// SIMATIC S7-200 project (STEP 7-Micro/WIN), CPU 221 REL 01.10

SYMBOL_TABLE USER1
BT               I0.0     // dieu khien bang tay
TD               I0.1     // dieu khien tu dong
s1               I0.2     // nut giu mo cong
s3               I0.3     // cong tac hanh trinh mo cong
s2               I0.4     // nut giu dong cong
s4               I0.5     // cong tac hanh trinh dong cong
open             I0.6     // mo cua o che do tu dong
close            I0.7     // dong cua o che do tu dong
s5               I1.0     // dung he thong
CDBT             Q0.0     // che do bang tay
CDTD             Q0.1     // che do tu dong
MT               Q0.2     // mo cong
MN               Q0.3     // dong cong
H1               Q0.4     // den bao
s6               I1.1     // dole nhiet dung he thong
END_SYMBOL_TABLE

ORGANIZATION_BLOCK MAIN:OB1
TITLE=PROGRAM COMMENTS
BEGIN
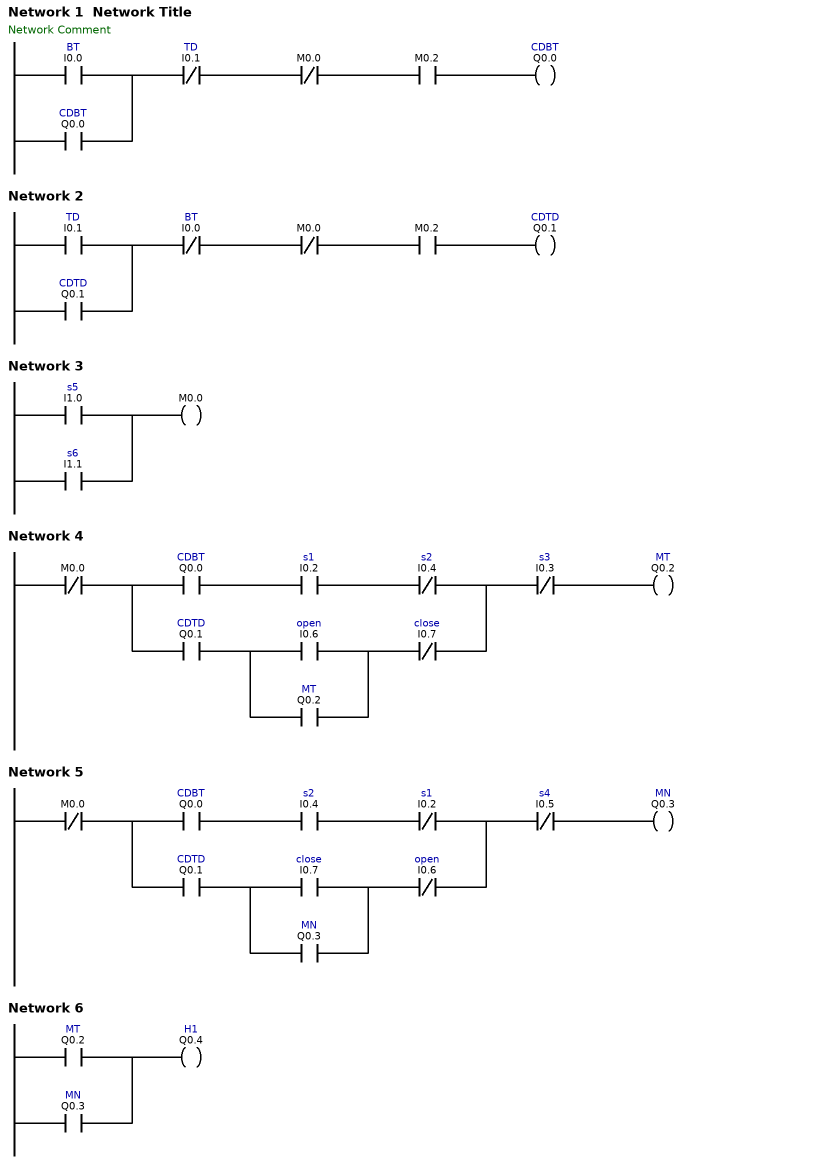
Network 1 // Network Title
// Network Comment
LD     BT:I0.0
O      CDBT:Q0.0
AN     TD:I0.1
AN     M0.0
A      M0.2
=      CDBT:Q0.0
Network 2
LD     TD:I0.1
O      CDTD:Q0.1
AN     BT:I0.0
AN     M0.0
A      M0.2
=      CDTD:Q0.1
Network 3
LD     s5:I1.0
O      s6:I1.1
=      M0.0
Network 4
LDN    M0.0
LD     CDBT:Q0.0
A      s1:I0.2
AN     s2:I0.4
LD     CDTD:Q0.1
LD     open:I0.6
O      MT:Q0.2
ALD
AN     close:I0.7
OLD
ALD
AN     s3:I0.3
=      MT:Q0.2
Network 5
LDN    M0.0
LD     CDBT:Q0.0
A      s2:I0.4
AN     s1:I0.2
LD     CDTD:Q0.1
LD     close:I0.7
O      MN:Q0.3
ALD
AN     open:I0.6
OLD
ALD
AN     s4:I0.5
=      MN:Q0.3
Network 6
LD     MT:Q0.2
O      MN:Q0.3
=      H1:Q0.4
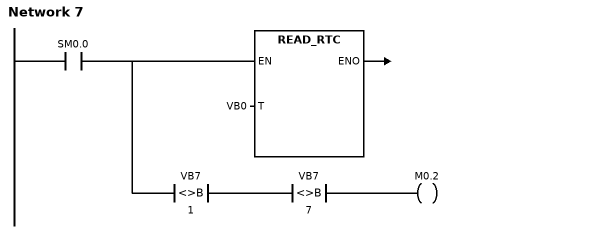
Network 7
LD     SM0.0
TODR   VB0
AB<>   VB7, 1
AB<>   VB7, 7
=      M0.2
END_ORGANIZATION_BLOCK
